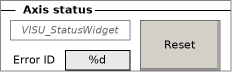
VISUALIZATION VISU_BaseAxis_Status  // 232x72
VAR_IN_OUT
	axis : BaseAxis;
    axisWidget : BaseAxisWidget;
END_VAR
    Label (20,0 75x20), "Axis status"
    Line (95,10) (230,10)
    Line (0,10) (15,10)
    Frame (10,20 120x20)
        shows VISU_StatusWidget(widget := axisWidget.actualStatus)
    Label (10,50 65x20), "Error ID"
    Rectangle (65,50 65x20), "%d", text variable: axis.axis_ref.Status.ErrorId
    Button (140,20 80x50), "Reset", input disabled if: axis.processes.reset.statuses.enabledStatus.disabled
        OnMouseClick: execute { axis.processes.reset.do_request := TRUE; }
END_VISUALIZATION

(* stored: Version 1.1.0.1, ProductVersion 3.1.4019.2
   Visu VISU_BaseAxis_Status: Id {acfc726c-0c42-4164-924a-edeff3922526} *)
